// TIA Portal project "DENEME_2022_06_27" (V16)

(* hardware
DEVICE "S71500/ET200MP station_1"  S7-1500 station
   slot 0: "Rail_0"  Rack  6ES7 590-1***0-0AA0
   slot 1: "PLC_1"  CPU 1512C-1 PN  6ES7 512-1CK01-0AB0  V2.8
      slot 3: "CPU display_1"  6ES7591-1AA00-0AA0
      slot 32768: "PROFINET interface_1"  X1
         slot 32769: "Port_1"  X1 P1
         slot 32770: "Port_2"  X1 P2
      slot 34817: "Virtual CP interface port_1"  Virtual CP interface port  Virtual CP interface port
DEVICE "HMI_1"  KTP1200 Basic PN
   slot 0: "HMI_1"  KTP1200 Basic PN  6AV2 123-2MB03-0AX0  16.0.0.0
   slot 1: "HMI_RT_1"  KTP1200 Basic PN  6AV2 123-2MB03-0AX0  16.0.0.0
   slot 5: "HMI_1.IE_CP_1"  PROFINET Interface  16.0.0.0
      slot 1: "PROFINET Interface_1"  PROFINET Interface
         slot 1: "Port_1"  Port
*)

// ===== PLC "PLC_1"  CPU 1512C-1 PN =====

VAR_GLOBAL   // PLC tag table "Default tag table"
   "0 POSITION" AT %M6.3 : Bool;
   "MANUEL MODE" AT %M6.4 : Bool;
   "AUTO MODE" AT %M6.5 : Bool;
   "START" AT %M6.6 : Bool;
   "STOP" AT %M6.7 : Bool;
   "FORWARD BUTTON" AT %M7.0 : Bool;
   "REVERSE BUTTON" AT %M7.1 : Bool;
   "VALVE BUTTON" AT %M7.2 : Bool;
   "SENSOR 1" AT %M8.2 : Bool;
   "SENSOR 2" AT %M8.3 : Bool;
   "SENSOR 3" AT %M8.4 : Bool;
   "COUNTER RESET" AT %M7.3 : Bool;
   "FORWARD MOTOR" AT %Q0.0 : Bool;
   "REVERSE MOTOR" AT %Q0.1 : Bool;
   "VALVE" AT %Q0.2 : Bool;
   "FORWARD MOTOR MEM" AT %M5.0 : Bool;
   "REVERSE MOTOR MEM" AT %M5.1 : Bool;
   "VALVE MEM" AT %M5.2 : Bool;
   "SR_LATCH" AT %M5.3 : Bool;
   "SENSOR 2 MEM" AT %M5.4 : Bool;
   "MANUEL MEM" AT %M5.5 : Bool;
   "AUTO MEM" AT %M5.6 : Bool;
   "STOP SYSTEM MEM" AT %M5.7 : Bool;
   "PULSE 2 MEM" AT %M6.0 : Bool;
   "FORWARD MOTOR MEM 2" AT %M6.1 : Bool;
   "VALVE MEM 2" AT %M6.2 : Bool;
   "SENSOR_2_ALARM" AT %M7.4 : Bool;
   "SENSOR_3_ALARM" AT %M7.5 : Bool;
   "SR_FOR_SENSOR_2" AT %M7.6 : Bool;
   "SR_FOR_SENSOR_3" AT %M7.7 : Bool;
   "NEG_TRIG" AT %M8.0 : Bool;
   "ACTIVATE_SENSOR_2_TIMERS" AT %M8.1 : Bool;
   "SENSOR_1_ALARM" AT %M8.5 : Bool;
   "SENSOR_3_SR" AT %M8.6 : Bool;
   "PULSE_T2_S1" AT %M8.7 : Bool;
   "PULSE_T2_S2" AT %M9.0 : Bool;
END_VAR

// folder: System blocks/Program resources

DATA_BLOCK "TIMER_1"   // DB1
{ S7_Optimized_Access := 'TRUE' }
AUTHOR : Simatic
FAMILY : IEC
NAME : IEC_TMR
VERSION : 1.0
// stored: InstanceOfName IEC_TIMER
"IEC_TIMER"
BEGIN
END_DATA_BLOCK

DATA_BLOCK "FULL_COUNTER"   // DB2
{ S7_Optimized_Access := 'TRUE' }
AUTHOR : Simatic
FAMILY : IEC
NAME : CNTR
VERSION : 1.0
// stored: InstanceOfName IEC_COUNTER
"IEC_COUNTER"
BEGIN
END_DATA_BLOCK

DATA_BLOCK "EMPTY_COUNTER"   // DB3
{ S7_Optimized_Access := 'TRUE' }
AUTHOR : Simatic
FAMILY : IEC
NAME : CNTR
VERSION : 1.0
// stored: InstanceOfName IEC_COUNTER
"IEC_COUNTER"
BEGIN
END_DATA_BLOCK

DATA_BLOCK "COUNTER_FOR_VALVE"   // DB4
{ S7_Optimized_Access := 'TRUE' }
AUTHOR : Simatic
FAMILY : IEC
NAME : CNTR
VERSION : 1.0
// stored: InstanceOfName IEC_COUNTER
"IEC_COUNTER"
BEGIN
END_DATA_BLOCK

DATA_BLOCK "TIMER_1_AT_SENSOR_2"   // DB5
{ S7_Optimized_Access := 'TRUE' }
AUTHOR : Simatic
FAMILY : IEC
NAME : IEC_TMR
VERSION : 1.0
// stored: InstanceOfName IEC_TIMER
"IEC_TIMER"
BEGIN
END_DATA_BLOCK

DATA_BLOCK "TIMER_2_AT_SENSOR_2"   // DB6
{ S7_Optimized_Access := 'TRUE' }
AUTHOR : Simatic
FAMILY : IEC
NAME : IEC_TMR
VERSION : 1.0
// stored: InstanceOfName IEC_TIMER
"IEC_TIMER"
BEGIN
END_DATA_BLOCK

DATA_BLOCK "TIMER_1_AT_SENSOR_1"   // DB7
{ S7_Optimized_Access := 'TRUE' }
AUTHOR : Simatic
FAMILY : IEC
NAME : IEC_TMR
VERSION : 1.0
// stored: InstanceOfName IEC_TIMER
"IEC_TIMER"
BEGIN
END_DATA_BLOCK

DATA_BLOCK "TIMER_2_AT_SENSOR_1"   // DB8
{ S7_Optimized_Access := 'TRUE' }
AUTHOR : Simatic
FAMILY : IEC
NAME : IEC_TMR
VERSION : 1.0
// stored: InstanceOfName IEC_TIMER
"IEC_TIMER"
BEGIN
END_DATA_BLOCK

DATA_BLOCK "ALARM_1_COUNTER"   // DB9
{ S7_Optimized_Access := 'TRUE' }
AUTHOR : Simatic
FAMILY : IEC
NAME : CNTR
VERSION : 1.0
// stored: InstanceOfName IEC_COUNTER
"IEC_COUNTER"
BEGIN
END_DATA_BLOCK

// folder: (top level)

FUNCTION "CALISMA" : Void   // FC1, LAD
{ S7_Optimized_Access := 'TRUE' }
VERSION : 0.1
   VAR_TEMP   // added for the SCL form of the ladder/FBD networks
      _w1 : Bool;
      _w2 : Bool;
      _w3 : Bool;
      _w4 : Bool;
   END_VAR
BEGIN

REGION Network 1: START-STOP AND SYSTEM MODE
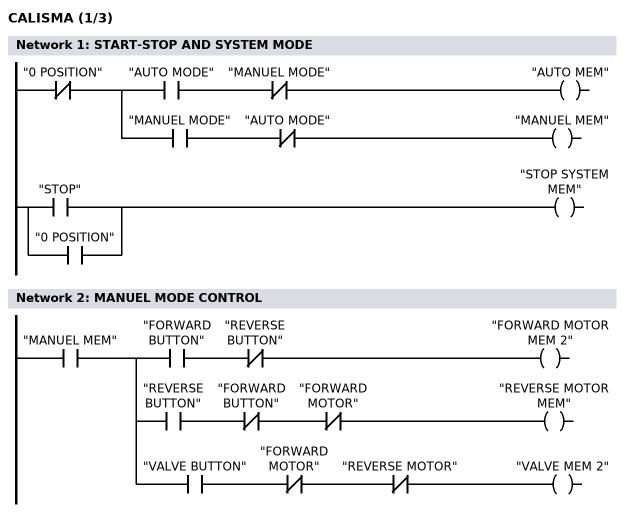
   RUNG wire#powerrail
      I_Contact( "0 POSITION" )
      wire#w1
      Contact( "AUTO MODE" )
      I_Contact( "MANUEL MODE" )
      Coil( "AUTO MEM" )
   END_RUNG
   RUNG wire#w1
      Contact( "MANUEL MODE" )
      I_Contact( "AUTO MODE" )
      Coil( "MANUEL MEM" )
   END_RUNG
   RUNG wire#powerrail
      Contact( "STOP" )
      wire#w2
      Coil( "STOP SYSTEM MEM" )
   END_RUNG
   RUNG wire#powerrail
      Contact( "0 POSITION" )
   END_RUNG wire#w2
   // the same network as SCL:
   "AUTO MEM" := NOT "0 POSITION" AND "AUTO MODE" AND NOT "MANUEL MODE";
   "MANUEL MEM" := NOT "0 POSITION" AND "MANUEL MODE" AND NOT "AUTO MODE";
   "STOP SYSTEM MEM" := "STOP" OR "0 POSITION";
END_REGION

REGION Network 2: MANUEL MODE CONTROL
   RUNG wire#powerrail
      Contact( "MANUEL MEM" )
      wire#w1
      Contact( "FORWARD BUTTON" )
      I_Contact( "REVERSE BUTTON" )
      Coil( "FORWARD MOTOR MEM 2" )
   END_RUNG
   RUNG wire#w1
      Contact( "REVERSE BUTTON" )
      I_Contact( "FORWARD BUTTON" )
      I_Contact( "FORWARD MOTOR" )
      Coil( "REVERSE MOTOR MEM" )
   END_RUNG
   RUNG wire#w1
      Contact( "VALVE BUTTON" )
      I_Contact( "FORWARD MOTOR" )
      I_Contact( "REVERSE MOTOR" )
      Coil( "VALVE MEM 2" )
   END_RUNG
   // the same network as SCL:
   "FORWARD MOTOR MEM 2" := "MANUEL MEM" AND "FORWARD BUTTON" AND NOT "REVERSE BUTTON";
   "REVERSE MOTOR MEM" := "MANUEL MEM" AND "REVERSE BUTTON" AND NOT "FORWARD BUTTON" AND NOT "FORWARD MOTOR";
   "VALVE MEM 2" := "MANUEL MEM" AND "VALVE BUTTON" AND NOT "FORWARD MOTOR" AND NOT "REVERSE MOTOR";
END_REGION

REGION Network 3: AUTO MODE CONTROL
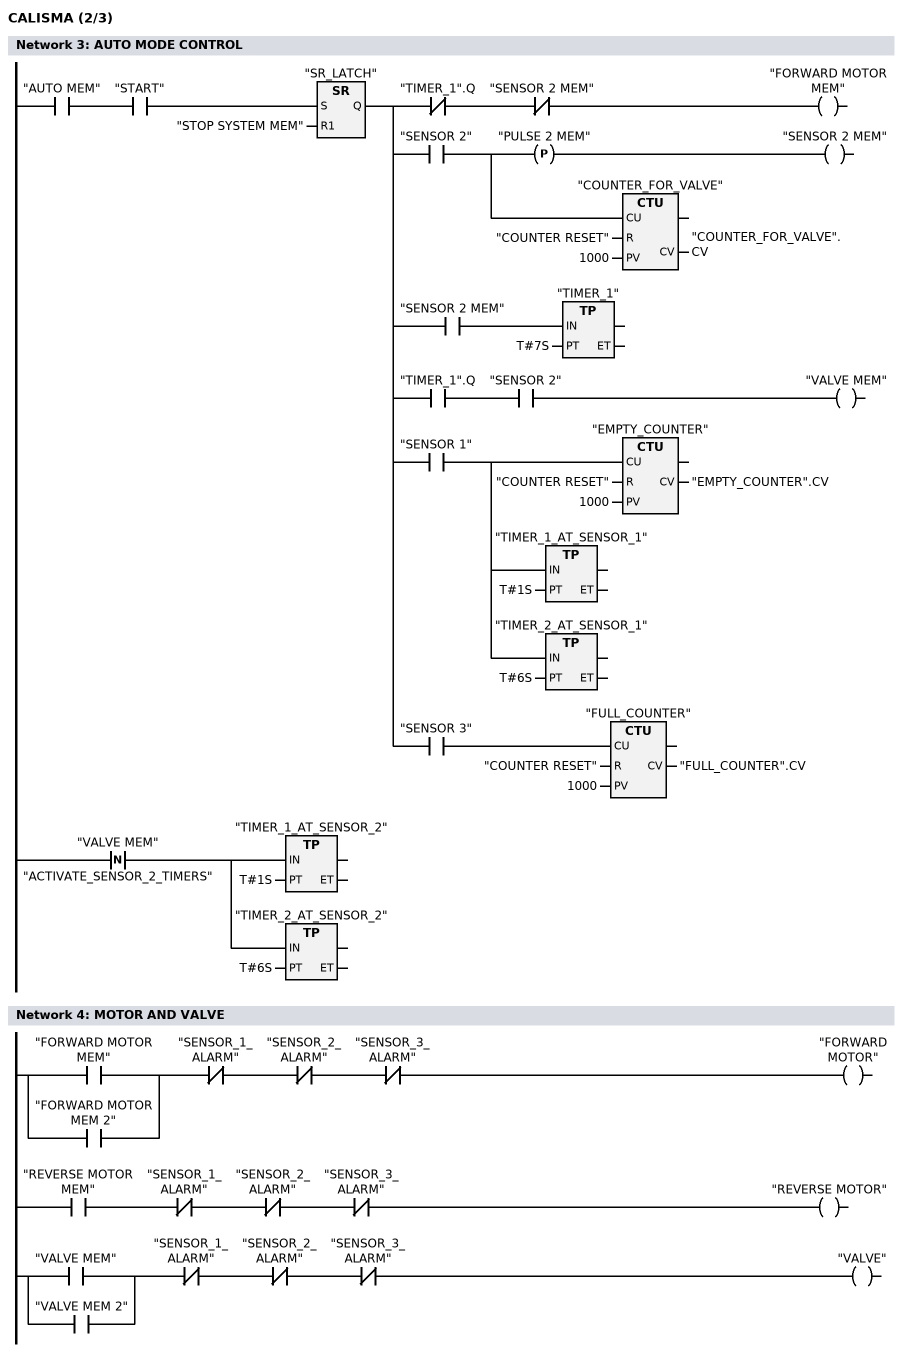
   IF "AUTO MEM" AND "START" THEN
       "SR_LATCH" := TRUE;   // SR flip-flop
   END_IF;
   IF "STOP SYSTEM MEM" THEN "SR_LATCH" := FALSE; END_IF;
   "FORWARD MOTOR MEM" := "SR_LATCH" AND NOT "TIMER_1".Q AND NOT "SENSOR 2 MEM";
   #_w1 := "SR_LATCH" AND "SENSOR 2";
   #_w2 := #_w1 AND NOT "PULSE 2 MEM";   // rising edge
   "PULSE 2 MEM" := #_w1;
   "SENSOR 2 MEM" := #_w2;
   "COUNTER_FOR_VALVE".CTU(CU := #_w1, R := "COUNTER RESET", PV := 1000, CV => "COUNTER_FOR_VALVE".CV);
   "TIMER_1".TP(IN := "SR_LATCH" AND "SENSOR 2 MEM", PT := T#7S);
   "VALVE MEM" := "SR_LATCH" AND "TIMER_1".Q AND "SENSOR 2";
   #_w3 := "SR_LATCH" AND "SENSOR 1";
   "EMPTY_COUNTER".CTU(CU := #_w3, R := "COUNTER RESET", PV := 1000, CV => "EMPTY_COUNTER".CV);
   "TIMER_1_AT_SENSOR_1".TP(IN := #_w3, PT := T#1S);
   "TIMER_2_AT_SENSOR_1".TP(IN := #_w3, PT := T#6S);
   "FULL_COUNTER".CTU(CU := "SR_LATCH" AND "SENSOR 3",
                      R := "COUNTER RESET",
                      PV := 1000,
                      CV => "FULL_COUNTER".CV);
   #_w4 := NOT "VALVE MEM" AND "ACTIVATE_SENSOR_2_TIMERS";   // falling edge of "VALVE MEM"
   "ACTIVATE_SENSOR_2_TIMERS" := "VALVE MEM";
   "TIMER_1_AT_SENSOR_2".TP(IN := #_w4, PT := T#1S);
   "TIMER_2_AT_SENSOR_2".TP(IN := #_w4, PT := T#6S);
END_REGION

REGION Network 4: MOTOR AND VALVE
   RUNG wire#powerrail
      Contact( "FORWARD MOTOR MEM" )
      wire#w1
      I_Contact( "SENSOR_1_ALARM" )
      I_Contact( "SENSOR_2_ALARM" )
      I_Contact( "SENSOR_3_ALARM" )
      Coil( "FORWARD MOTOR" )
   END_RUNG
   RUNG wire#powerrail
      Contact( "FORWARD MOTOR MEM 2" )
   END_RUNG wire#w1
   RUNG wire#powerrail
      Contact( "REVERSE MOTOR MEM" )
      I_Contact( "SENSOR_1_ALARM" )
      I_Contact( "SENSOR_2_ALARM" )
      I_Contact( "SENSOR_3_ALARM" )
      Coil( "REVERSE MOTOR" )
   END_RUNG
   RUNG wire#powerrail
      Contact( "VALVE MEM" )
      wire#w2
      I_Contact( "SENSOR_1_ALARM" )
      I_Contact( "SENSOR_2_ALARM" )
      I_Contact( "SENSOR_3_ALARM" )
      Coil( "VALVE" )
   END_RUNG
   RUNG wire#powerrail
      Contact( "VALVE MEM 2" )
   END_RUNG wire#w2
   // the same network as SCL:
   "FORWARD MOTOR" := ("FORWARD MOTOR MEM" OR "FORWARD MOTOR MEM 2") AND NOT "SENSOR_1_ALARM" AND NOT "SENSOR_2_ALARM" AND NOT "SENSOR_3_ALARM";
   "REVERSE MOTOR" := "REVERSE MOTOR MEM" AND NOT "SENSOR_1_ALARM" AND NOT "SENSOR_2_ALARM" AND NOT "SENSOR_3_ALARM";
   "VALVE" := ("VALVE MEM" OR "VALVE MEM 2") AND NOT "SENSOR_1_ALARM" AND NOT "SENSOR_2_ALARM" AND NOT "SENSOR_3_ALARM";
END_REGION

REGION Network 5: ALARM
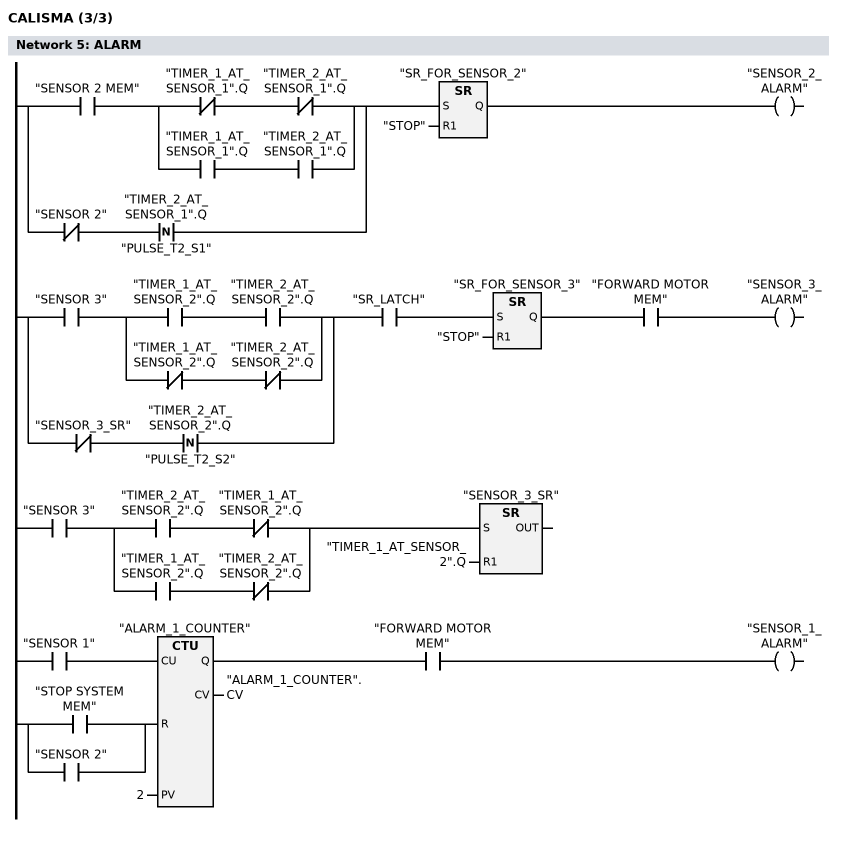
   #_w1 := NOT "SENSOR 2" AND NOT "TIMER_2_AT_SENSOR_1".Q AND "PULSE_T2_S1";   // falling edge of "TIMER_2_AT_SENSOR_1".Q
   "PULSE_T2_S1" := "TIMER_2_AT_SENSOR_1".Q;
   IF ("SENSOR 2 MEM" AND ((NOT "TIMER_1_AT_SENSOR_1".Q AND NOT "TIMER_2_AT_SENSOR_1".Q) OR ("TIMER_1_AT_SENSOR_1".Q AND "TIMER_2_AT_SENSOR_1".Q))) OR #_w1 THEN
       "SR_FOR_SENSOR_2" := TRUE;   // SR flip-flop
   END_IF;
   IF "STOP" THEN "SR_FOR_SENSOR_2" := FALSE; END_IF;
   "SENSOR_2_ALARM" := "SR_FOR_SENSOR_2";
   #_w2 := NOT "SENSOR_3_SR" AND NOT "TIMER_2_AT_SENSOR_2".Q AND "PULSE_T2_S2";   // falling edge of "TIMER_2_AT_SENSOR_2".Q
   "PULSE_T2_S2" := "TIMER_2_AT_SENSOR_2".Q;
   IF (("SENSOR 3" AND (("TIMER_1_AT_SENSOR_2".Q AND "TIMER_2_AT_SENSOR_2".Q) OR (NOT "TIMER_1_AT_SENSOR_2".Q AND NOT "TIMER_2_AT_SENSOR_2".Q))) OR #_w2) AND "SR_LATCH" THEN
       "SR_FOR_SENSOR_3" := TRUE;   // SR flip-flop
   END_IF;
   IF "STOP" THEN "SR_FOR_SENSOR_3" := FALSE; END_IF;
   "SENSOR_3_ALARM" := "SR_FOR_SENSOR_3" AND "FORWARD MOTOR MEM";
   IF "SENSOR 3" AND (("TIMER_2_AT_SENSOR_2".Q AND NOT "TIMER_1_AT_SENSOR_2".Q) OR ("TIMER_1_AT_SENSOR_2".Q AND NOT "TIMER_2_AT_SENSOR_2".Q)) THEN
       "SENSOR_3_SR" := TRUE;   // SR flip-flop
   END_IF;
   IF "TIMER_1_AT_SENSOR_2".Q THEN "SENSOR_3_SR" := FALSE; END_IF;
   "ALARM_1_COUNTER".CTU(CU := "SENSOR 1",
                         R := "STOP SYSTEM MEM" OR "SENSOR 2",
                         PV := 2,
                         CV => "ALARM_1_COUNTER".CV);
   "SENSOR_1_ALARM" := "ALARM_1_COUNTER".Q AND "FORWARD MOTOR MEM";
END_REGION
END_FUNCTION

ORGANIZATION_BLOCK "Main"   // OB1, LAD, ProgramCycle
TITLE = "Main Program Sweep (Cycle)"
{ S7_Optimized_Access := 'TRUE' }
VERSION : 0.1
   VAR_INPUT
      Initial_Call : Bool;   // Initial call of this OB
      Remanence : Bool;   // =True, if remanent data are available
   END_VAR
BEGIN

REGION Network 1
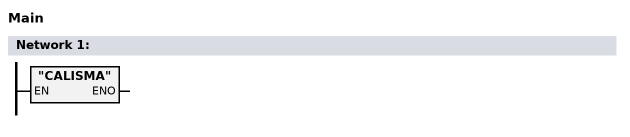
   RUNG wire#powerrail
      "CALISMA"()
   END_RUNG
   // the same network as SCL:
   "CALISMA"();
END_REGION
END_ORGANIZATION_BLOCK

(* ===== HMI "HMI_RT_1" =====
system functions are stored by id; their names below are inferred from use
connection "HMI_Connection_1": ETHERNET, SMART_S7_1500_OMS

HMI tags "Default tag table"
   "0 POSITION" : Bool = PLC "0 POSITION" AT %M6.3, 1 s
   "MANUEL MODE" : Bool = PLC "MANUEL MODE" AT %M6.4, 1 s
   "AUTO MODE" : Bool = PLC "AUTO MODE" AT %M6.5, 1 s
   "START" : Bool = PLC START AT %M6.6, 1 s
   "STOP" : Bool = PLC STOP AT %M6.7, 1 s
   "FORWARD BUTTON" : Bool = PLC "FORWARD BUTTON" AT %M7.0, 1 s
   "REVERSE BUTTON" : Bool = PLC "REVERSE BUTTON" AT %M7.1, 1 s
   "VALVE BUTTON" : Bool = PLC "VALVE BUTTON" AT %M7.2, 1 s
   "SENSOR 1" : Bool = PLC "SENSOR 1" AT %M8.2, 1 s
   "SENSOR 2" : Bool = PLC "SENSOR 2" AT %M8.3, 1 s
   "SENSOR 3" : Bool = PLC "SENSOR 3" AT %M8.4, 1 s
   "COUNTER RESET" : Bool = PLC "COUNTER RESET" AT %M7.3, 1 s
   "FORWARD MOTOR" : Bool = PLC "FORWARD MOTOR" AT %Q0.0, 1 s
   "REVERSE MOTOR" : Bool = PLC "REVERSE MOTOR" AT %Q0.1, 1 s
   "VALVE" : Bool = PLC VALVE AT %Q0.2, 1 s
   "FORWARD MOTOR MEM" : Bool = PLC "FORWARD MOTOR MEM" AT %M5.0, 1 s
   "REVERSE MOTOR MEM" : Bool = PLC "REVERSE MOTOR MEM" AT %M5.1, 1 s
   "VALVE MEM" : Bool = PLC "VALVE MEM" AT %M5.2, 1 s
   "SR_LATCH" : Bool = PLC SR_LATCH AT %M5.3, 1 s
   "SENSOR 2 MEM" : Bool = PLC "SENSOR 2 MEM" AT %M5.4, 1 s
   "MANUEL MEM" : Bool = PLC "MANUEL MEM" AT %M5.5, 1 s
   "AUTO MEM" : Bool = PLC "AUTO MEM" AT %M5.6, 1 s
   "STOP SYSTEM MEM" : Bool = PLC "STOP SYSTEM MEM" AT %M5.7, 1 s
   "PULSE 2 MEM" : Bool = PLC "PULSE 2 MEM" AT %M6.0, 1 s
   "EMPTY COUNTER" : Int = PLC EMPTY_COUNTER.CV AT %DB1.DBX0.0, 1 s
   "FULL COUNTER" : Int = PLC FULL_COUNTER.CV AT %DB1.DBW0, 1 s
   "TIMER" : Time = PLC TIMER_1.ET AT %DB1.DBW0, 1 s
   "SENSOR_2_ALARM" : Bool = PLC SENSOR_2_ALARM AT %M7.4, 1 s
   "SENSOR_3_ALARM" : Bool = PLC SENSOR_3_ALARM AT %M7.5, 1 s
   "SENSOR_1_ALARM" : Bool = PLC SENSOR_1_ALARM AT %M8.5, 1 s

screen "Root screen" 1280x800, template "Template_1"
   Circle "Circle_1" at 29,40 size 24x24
      Appearance <- "SENSOR 1"
   Circle "Circle_2" at 94,40 size 24x24
      Appearance <- "SENSOR 2"
   Circle "Circle_3" at 163,40 size 24x24
      Appearance <- "SENSOR 3"
   TextField "Text field_1" at 9,22 size 69x18; Text 'SENSOR 1'
   TextField "Text field_2" at 76,22 size 69x18; Text 'SENSOR 2'
   TextField "Text field_3" at 143,22 size 69x18; Text 'SENSOR 3'
   Button "Button_1" at 1156,41 size 103x35; TextOff 'FORWARD MOTOR'
      on Press: function_b14e0dd5("FORWARD BUTTON", 0)
      Appearance <- "FORWARD MOTOR"
   Button "Button_2" at 1161,92 size 103x35; TextOff 'REVERSE MOTOR'
      Appearance <- "REVERSE MOTOR MEM"
      on Press: function_b14e0dd5("REVERSE BUTTON", 0)
   Button "Button_3" at 1161,144 size 103x35; TextOff 'VALVE'
      Appearance <- "VALVE"
      on Press: function_b14e0dd5("VALVE BUTTON", 0)
   Button "Button_4" at 1032,40 size 103x35; TextOff 'START'
      Appearance <- "START"
      on Press: function_b14e0dd5("START", 0)
   Button "Button_5" at 1032,92 size 103x35; TextOff 'STOP'
      Appearance <- "STOP"
      on Press: function_b14e0dd5("STOP", 0)
   Button "Button_6" at 1032,144 size 103x35; TextOff 'COUNTER RESET'
      Appearance <- "COUNTER RESET"
      on Press: function_b14e0dd5("COUNTER RESET", 0)
   Switch "Switch_1" at 1164,348 size 64x32; CaptionText 'Switch'; TextOff 'ON'; TextOn 'OFF'
      Appearance <- "0 POSITION"
      on SwitchOn: SetBit("0 POSITION")
      on SwitchOff: ResetBit("0 POSITION")
      ProcessValue <- "0 POSITION"
   Switch "Switch_2" at 1164,414 size 64x32; TextOn 'ON'; CaptionText 'Switch'; TextOff 'OFF'
      on SwitchOn: SetBit("AUTO MODE")
      on SwitchOff: ResetBit("AUTO MODE")
      Appearance <- "AUTO MODE"
      ProcessValue <- "AUTO MODE"
   Switch "Switch_3" at 1164,480 size 64x32; TextOn 'ON'; CaptionText 'Switch'; TextOff 'OFF'
      Appearance <- "MANUEL MODE"
      on SwitchOn: SetBit("MANUEL MODE")
      on SwitchOff: ResetBit("MANUEL MODE")
      ProcessValue <- "MANUEL MODE"
   TextField "Text field_4" at 1146,331 size 100x17; Text 'SYSTEM ON/OFF'
   TextField "Text field_5" at 1157,397 size 78x17; Text 'AUTO MODE'
   TextField "Text field_6" at 1151,463 size 92x17; Text 'MANUEL MODE'
   Bar "Bar_1" at 290,40 size 100x200; MinimumValue 0; MaximumValue 100
      ProcessValue <- "EMPTY COUNTER"
      Appearance <- "EMPTY COUNTER"
   Bar "Bar_2" at 450,40 size 100x200; MinimumValue 0; MaximumValue 100
      ProcessValue <- "FULL COUNTER"
      Appearance <- "FULL COUNTER"
   TextField "Text field_7" at 275,15 size 132x25; Text 'EMPTY BOTTLE'
   TextField "Text field_8" at 440,15 size 118x25; Text 'FULL BOTTLE'
   IOField "I/O field_1" at 243,722 size 96x32; FormatPattern s9999999999
      ProcessValue <- "TIMER"
      Appearance <- "TIMER"
   TextField "Text field_9" at 231,693 size 119x25; Text 'VALVE TIMER'
   Circle "Circle_4" at 53,610 size 48x48
      Appearance <- "FORWARD MOTOR"
   Circle "Circle_5" at 269,610 size 48x48
      Appearance <- "REVERSE MOTOR"
   TextField "Text field_10" at 9,585 size 162x25; Text 'FORWARD MOTOR'
   TextField "Text field_11" at 220,585 size 149x25; Text 'REVERSE MOTOR'
   Rectangle "Rectangle_1" at 37,718 size 78x34
      Appearance <- "VALVE"
   TextField "Text field_12" at 42,692 size 59x25; Text 'VALVE'
   Circle "Circle_6" at 52,179 size 24x24
      Appearance <- "SENSOR_2_ALARM"
   Circle "Circle_7" at 54,237 size 24x24
      Appearance <- "SENSOR_3_ALARM"
   TextField "Text field_13" at 14,155 size 101x17; Text 'ALARM SENSOR 2'
   TextField "Text field_14" at 18,215 size 101x17; Text 'ALARM SENSOR 3'
   Button "Button_7" at 20,286 size 99x36; TextOff 'SENSOR 1 INPUT'
      Appearance <- "SENSOR 1"
      on Press: function_b14e0dd5("SENSOR 1", 0)
   Button "Button_8" at 20,344 size 99x36; TextOff 'SENSOR 2 INPUT'
      Appearance <- "SENSOR 2"
      on Press: function_b14e0dd5("SENSOR 2", 0)
   Button "Button_9" at 20,402 size 99x36; TextOff 'SENSOR 3 INPUT'
      Appearance <- "SENSOR 3"
      on Press: function_b14e0dd5("SENSOR 3", 0)
   Circle "Circle_8" at 54,118 size 24x24
      Appearance <- "SENSOR_1_ALARM"
   TextField "Text field_15" at 14,92 size 101x17; Text 'ALARM SENSOR 1'
*)